Fanuc KAREL source: CA0106.KL

-- PROVISIONAL review KL for V940-1; original PC SHA256 e60b756f62dab9f14bd2808bd1ed4c249810d73d2e7ae2cc0e48af2b2477be7c
-- Incomplete behavior may be omitted. Consult companion uncertainty JSON. Do not deploy.
PROGRAM CA0106
%NOLOCKGROUP
BEGIN
  -- V9_ZERO_TABLE_METADATA_HINT layout=0001; no indexed target words; source/name/runtime held
  -- UNRESOLVED_PC offsets 0-1; opcodes 7B
  -- UNRESOLVED_PC offsets 6-22; opcodes 2D,2E,69,7F
  -- UNRESOLVED_PC offsets 27-31; opcodes 7F
  -- UNRESOLVED_PC offsets 36-43; opcodes 9C,23
  -- UNRESOLVED_PC offsets 48-55; opcodes 9D,23
  -- UNRESOLVED_PC offsets 60-71; opcodes 2E,23
  -- UNRESOLVED_PC offsets 76-83; opcodes 9D,23
  -- UNRESOLVED_PC offsets 88-97; opcodes 3F,75
  -- UNRESOLVED_PC offsets 102-116; opcodes 2E,22,9D,33,35
  -- UNRESOLVED_PC offsets 121-135; opcodes 2E,22,9D,33,35
  -- UNRESOLVED_PC offsets 140-155; opcodes 2E,22,32,35
  -- UNRESOLVED_PC offsets 160-175; opcodes 2E,22,32,35
  -- UNRESOLVED_PC offsets 180-196; opcodes 27,22,AA,23
  -- UNRESOLVED_PC offsets 201-205; opcodes 7F
END CA0106
